   (*процесс*)
   IF "Technology".Regim = 11 THEN
       CASE "Technology".Regim_plan_stop_step OF
           0:  //плавный вывод ЗРГ на значение минимальной мощности ПИД регулятором
               IF "Sensors".ZRG_middle.Value THEN
                   "Control_ZRG".Mode := TRUE;
                   "Control_ZRG".Mode_from_PLC := TRUE;
                   IF "Control_ZRG".SP_PID > 10.0 THEN
                       "Control_ZRG".SP_PID := "Control_ZRG".SP_PID - 0.001;
                   END_IF;
               ELSE
                   //переход на следующий шаг
                   "Technology".Regim_plan_stop_step := 1;
               END_IF;

           1:  //Контроль достижения минимальной мощности
                   //снимаем защиту Понижение давления газа перед горелкой
                   "Alarms_and_warnings".Enable_Alarm_P_gas_before_burner_min := FALSE;
                   //снимаем защиту Повышение давления газа перед горелкой
                   "Alarms_and_warnings".Enable_Alarm_P_gas_before_burner_max := FALSE;
                   //отключаем ПИД регулирование ЗРГ
                   "Control_ZRG".Mode_from_PLC := FALSE;
                   "Control_ZRG".Manual_close_from_PLC := FALSE;
                   "Control_ZRG".Manual_open_from_PLC := FALSE;
                   //переход на следующий шаг
                   "Technology".Regim_plan_stop_step := 2;

           2:  //снимаем защиту Понижение давления сетевой воды за котлом
               "Alarms_and_warnings".Enable_Alarm_P_water_after_boiler_min := FALSE;
               //снимаем защиту Повышение давления сетевой воды за котлом
               "Alarms_and_warnings".Enable_Alarm_P_water_after_boiler_max := FALSE;
               //снимаем защиту Повышение температуры сетевой воды за котлом
               "Alarms_and_warnings".Enable_Alarm_T_water_after_boiler_max := FALSE;
               //снимаем защиту Понижение расхода сетевой воды через котел
               "Alarms_and_warnings".Enable_Alarm_Q_water_boiler_min := FALSE;

               //снимаем защиту Невоспламенение или погасание факела горелки котла
               "Alarms_and_warnings".Enable_Alarm_Not_flame_burner := FALSE;

               //перевод газовых исполнительных механизмов в исходное состояние
               "Control_PZK1".Mode := TRUE;    //закрываем ПЗК1
               "Control_PZK1".Avto_open := FALSE;
               "Control_PZK2".Mode := TRUE;    //закрываем ПЗК2
               "Control_PZK2".Avto_open := FALSE;
               "Control_KO".Mode := TRUE;  //закрываем КО
               "Control_KO".Avto_open := FALSE;
               "Control_KZ".Mode := TRUE;  //закрываем КЗ
               "Control_KZ".Avto_open := FALSE;
               "Control_KB".Mode := TRUE;  //открываем КБ
               "Control_KB".Avto_close := FALSE;
               "Control_IVN".Mode := TRUE; //отключаем ИВН
               "Control_IVN".Avto_on := FALSE;

               //перевод регуляторов разряжения и вентиляции на вентиляционные параметры
               IF "Sensors".DS_invertor_mode.Value THEN
                   "Control_DS".Mode := TRUE;
                   "Control_DS".Mode_from_PLC := TRUE;
                   "Control_DS".SP_PID := "RegMap".dP_furnace_ventilation;
               END_IF;
               IF "Sensors".DS_powergrid_mode.Value THEN
                   "Control_NAD".Mode := TRUE;
                   "Control_NAD".Mode_from_PLC := TRUE;
                   "Control_NAD".SP_PID := "RegMap".dP_furnace_ventilation;
               END_IF;
               IF "Sensors".DV_invertor_mode.Value THEN
                   "Control_DV".Mode := TRUE;
                   "Control_DV".Mode_from_PLC := TRUE;
                   "Control_DV".SP_PID := "RegMap".P_air_ventilation;
               END_IF;
               IF "Sensors".DV_powergrid_mode.Value THEN
                   "Control_NAV".Mode := TRUE;
                   "Control_NAV".Mode_from_PLC := TRUE;
                   "Control_NAV".SP_PID := "RegMap".P_air_ventilation;
               END_IF;

               //запускаем контрольный таймер
               "Timer".PLAN_STOP_temp_PT := T#60s;
               "Timer".PLAN_STOP_temp_IN := TRUE;
               //проверяем положение ИМ по газу
               IF NOT "Sensors".PZK1_open.Value AND
                   NOT "Sensors".PZK2_not_close.Value AND
                   NOT "Sensors".KO_open.Value AND
                   NOT "Sensors".KZ_open.Value AND
                   NOT "Sensors".KB_close.Value THEN
                   //переход далее
                   "Timer".PLAN_STOP_temp_IN := FALSE;
                   "Message".PLAN_STOP_not_initial_state_gas := FALSE;
                   "Technology".Regim_plan_stop_step := 3;
               END_IF;
               //если контрольное время вышло
               IF "Timer".PLAN_STOP_temp_Q THEN
                   "Message".PLAN_STOP_not_initial_state_gas := TRUE;
               END_IF;

           3:  //задержка 6 сек
               "Timer".PLAN_STOP_temp_PT := T#6s;
               "Timer".PLAN_STOP_temp_IN := TRUE;
               //переход далее
               IF "Timer".PLAN_STOP_temp_Q THEN
                   "Timer".PLAN_STOP_temp_IN := FALSE;
                   //переход на режим ПОСТОСТАНОВОЧНАЯ ОПРЕССОВКА
                   "Technology".Regim := 12;
               END_IF;
           ELSE
               "Technology".Regim_plan_stop_step := 0;
       END_CASE;
   ELSE
       //Сброс текущего шага
       "Technology".Regim_plan_stop_step := 0;
       //Сброс всех сообщений по данному режиму
       "Message".PLAN_STOP_not_initial_state_gas := FALSE;
       //сброс таймеров
       "Timer".PLAN_STOP_temp_IN := FALSE;
   END_IF;
END_FUNCTION

FUNCTION "Regim_STOP_PRESS" : Void   // FC22, SCL
{ S7_Optimized_Access := 'TRUE' }
VERSION : 0.1
BEGIN
   (*Режим ПОСТОСТАНОВОЧНАЯ ОПРЕССОВКА*)
   (*таймеры*)
   "Timer_STOP_PRESS_temp_DB".TON(IN := "Timer".STOP_PRESS_temp_IN,
                                  PT := "Timer".STOP_PRESS_temp_PT,
                                  Q => "Timer".STOP_PRESS_temp_Q);
   (*процесс*)
   IF "Technology".Regim = 12 THEN
       IF ("Sensors".DV_invertor_on.Value OR "Sensors".DV_powergrid_on.Value) AND
           ("Sensors".DS_invertor_on.Value OR "Sensors".DS_powergrid_on.Value) THEN
           CASE "Technology".Regim_stop_press_step OF
               0:  //анализ разрешения постостановочной опрессовки
                   IF "Technology".Stop_press_enable AND (NOT "Technology".Ventilation_conducted OR "Technology".transition_ignition) THEN
                       //переход на следующий шаг
                       "Technology".Regim_stop_press_step := 1;
                   ELSE
                       //переход на режим УКОРОЧЕННАЯ ВЕНТИЛЯЦИЯ
                       "Technology".Regim := 13;
                   END_IF;

               1:  //контроль положения исполнительных механизмов по газу
                   IF NOT "Sensors".PZK1_open.Value AND
                       NOT "Sensors".PZK2_not_close.Value AND
                       NOT "Sensors".KO_open.Value AND
                       NOT "Sensors".KZ_open.Value AND
                       NOT "Sensors".KB_close.Value THEN
                       //переход на следующий шаг
                       "Technology".Regim_stop_press_step := 2;
                   END_IF;

               2:  //контроль min P 
                   IF "Sensors".P_gas_before_PZK1_and_PZK2.Value < "Technology".SP_P_between_PZK_check_min THEN
                       //переход на следующий шаг
                       "Technology".Regim_stop_press_step := 3;
                   ELSE
                       "Message".STOP_PRESS_PZK1_or_KO_untight := TRUE;
                       "Technology".Regim_stop_press_step := 8;
                   END_IF;

               3:  //контроль max P
                   IF "Sensors".P_gas_before_PZK1_and_PZK2.Value < "Technology".SP_P_between_PZK_check_max THEN
                       //переход на следующий шаг
                       "Technology".Regim_stop_press_step := 4;
                   ELSE
                       "Message".STOP_PRESS_PZK1_or_KO_untight := TRUE;
                       "Technology".Regim_stop_press_step := 8;
                   END_IF;

               4:  //закрываем КБ
                   "Control_KB".Mode := TRUE;
                   "Control_KB".Avto_close := TRUE;
                   //контроль положения
                   IF "Sensors".KB_close.Value THEN
                       //переход на следующий шаг
                       "Timer".STOP_PRESS_temp_IN := FALSE;
                       "Technology".Regim_stop_press_step := 5;
                   END_IF;

               5:  //контроль отсутствия давления газа м/у ПЗК в течении заданного времени
                   "Timer".STOP_PRESS_temp_PT := T_CONV(INT_TO_DINT("Technology".SP_TIME_check_P_stop_press_min) * 1000);
                   "Timer".STOP_PRESS_temp_IN := TRUE;
                   IF "Timer".STOP_PRESS_temp_Q THEN
                       //переход на следующий шаг
                       "Timer".STOP_PRESS_temp_IN := FALSE;
                       "Technology".Regim_stop_press_step := 6;
                   ELSE
                       //если давление не в норме
                       IF ("Sensors".P_gas_before_PZK1_and_PZK2.Value > "Technology".SP_P_between_PZK_check_min) OR
                           ("Sensors".P_gas_before_PZK1_and_PZK2.Value > "Technology".SP_P_between_PZK_check_max) THEN
                           "Message".STOP_PRESS_PZK1_or_KO_untight := TRUE;
                           "Timer".STOP_PRESS_temp_IN := FALSE;
                           "Technology".Regim_stop_press_step := 8;
                       END_IF;
                   END_IF;

               6:  //открываем КО
                   "Control_KO".Mode := TRUE;
                   "Control_KO".Avto_open := TRUE;
                   IF "Sensors".KO_open.Value THEN
                       //переход на следующий шаг
                       "Timer".STOP_PRESS_temp_IN := FALSE;
                       "Technology".Regim_stop_press_step := 7;
                   END_IF;

               7:  //контроль достижения давления газа м/у ПЗК в течении заданного времени
                   "Timer".STOP_PRESS_temp_PT := T_CONV(INT_TO_DINT("Technology".SP_TIME_check_P_stop_press_max) * 1000);
                   "Timer".STOP_PRESS_temp_IN := TRUE;
                   IF "Timer".STOP_PRESS_temp_Q THEN
                       IF "Sensors".P_gas_before_BG_min.Value THEN
                           "Message".STOP_PRESS_P_before_BG_min := TRUE;
                       ELSE
                           "Message".STOP_PRESS_PZK2_or_KB_untight := TRUE;
                       END_IF;
                       "Timer".STOP_PRESS_temp_IN := FALSE;
                       "Technology".Regim_stop_press_step := 8;
                   ELSE
                       IF "Sensors".P_gas_before_PZK1_and_PZK2.Value > "Technology".SP_P_between_PZK_check_min THEN
                           //переход на следующий шаг
                           "Timer".STOP_PRESS_temp_IN := FALSE;
                           "Technology".Regim_stop_press_step := 8;
                       END_IF;
                   END_IF;

               8:  //закраваем КО
                   "Control_KO".Mode := TRUE;
                   "Control_KO".Avto_open := FALSE;
                   IF NOT "Sensors".KO_open.Value THEN
                       //переход на следующий шаг
                       "Technology".Regim_stop_press_step := 9;
                   END_IF;

               9:  //открываем КБ
                   "Control_KB".Mode := TRUE;
                   "Control_KB".Avto_close := FALSE;
                   IF NOT "Sensors".KB_close.Value THEN
                       //переход на следующий шаг
                       "Technology".Regim_stop_press_step := 10;
                   END_IF;

               10: //если опрессовка не прошла
                   IF "Message".STOP_PRESS_PZK1_or_KO_untight OR
                       "Message".STOP_PRESS_PZK2_or_KB_untight OR
                       "Message".STOP_PRESS_P_before_BG_min THEN
                       //переход на следующий шаг
                       "Timer".STOP_PRESS_temp_IN := FALSE;
                       "Technology".Regim_stop_press_step := 11;
                   ELSE
                       //если опрессовка успешно проведена
                       "Message".STOP_PRESS_success := TRUE;
                       //переход на следующий шаг
                       "Timer".STOP_PRESS_temp_IN := FALSE;
                       "Technology".Regim_stop_press_step := 11;
                   END_IF;

               11: //ожидание 5 сек
                   "Timer".STOP_PRESS_temp_PT := T#5s;
                   "Timer".STOP_PRESS_temp_IN := TRUE;
                   IF "Timer".STOP_PRESS_temp_Q THEN
                       "Timer".STOP_PRESS_temp_IN := FALSE;
                       "Message".STOP_PRESS_success := FALSE;
                       //переход на УКОРОЧЕННАЯ ВЕНТИЛЯЦИЯ
                       "Technology".Regim := 13;
                   END_IF;
               ELSE
                   "Technology".Regim_stop_press_step := 0;
           END_CASE;
       ELSE
           //перевод всех клапанов в исходное состояние
           "Control_PZK1".Mode := TRUE;        //закрываем ПЗК1
           "Control_PZK1".Avto_open := FALSE;
           "Control_PZK2".Mode := TRUE;        //закрываем ПЗК2
           "Control_PZK2".Avto_open := FALSE;
           "Control_KZ".Mode := TRUE;          //закрываем КЗ
           "Control_KZ".Avto_open := FALSE;
           "Control_KO".Mode := TRUE;          //закрываем КО
           "Control_KO".Avto_open := FALSE;
           "Control_KB".Mode := TRUE;          //открываем КБ
           "Control_KB".Avto_close := FALSE;
           "Control_IVN".Mode := TRUE;         //отключаем ИВН
           "Control_IVN".Avto_on := FALSE;
           //проверяем положение ИМ по газу
           IF NOT "Sensors".KB_close.Value AND //КБ открыт
               NOT "Sensors".KZ_open.Value AND //КЗ закрыт
               NOT "Sensors".KO_open.Value AND //КО закрыт
               NOT "Sensors".PZK1_open.Value AND   //ПЗК1 закрыт
               NOT "Sensors".PZK2_not_close.Value THEN  //ПЗК2 закрыт
               //переход далее
               //переход на УКОРОЧЕННАЯ ВЕНТИЛЯЦИЯ
               "Technology".Regim := 13;
           END_IF;
       END_IF;
   ELSE
       //сброс текущего шага
       "Technology".Regim_stop_press_step := 0;
       //сброс сообщений
       "Message".STOP_PRESS_PZK1_or_KO_untight := FALSE;
       "Message".STOP_PRESS_PZK2_or_KB_untight := FALSE;
       "Message".STOP_PRESS_P_before_BG_min := FALSE;
       "Message".STOP_PRESS_success := FALSE;
       //сброс таймеров
       "Timer".STOP_PRESS_temp_IN := FALSE;
   END_IF;
END_FUNCTION

FUNCTION "Regim_SHORT_VENTILATION" : Void   // FC23, SCL
{ S7_Optimized_Access := 'TRUE' }
VERSION : 0.1
BEGIN
   (*Режим УКОРОЧЕННАЯ ВЕНТИЛЯЦИЯ*)
   (*таймеры*)
   "Timer_SHORT_VENTILATION_temp_DB".TON(IN := "Timer".SHORT_VENTILATION_temp_IN,
                                         PT := "Timer".SHORT_VENTILATION_temp_PT,
                                         Q => "Timer".SHORT_VENTILATION_temp_Q);
   (*процесс*)
   IF "Technology".Regim = 13 THEN
       //снимаем защиту Повышение давления газа перед БГ
       "Alarms_and_warnings".Enable_Alarm_P_gas_before_BG_max := FALSE;
       //снимаем защиту Понижение давления газа перед БГ
       "Alarms_and_warnings".Enable_Alarm_P_gas_before_BG_min := FALSE;
       //закрываем ЗДГ
       "Control_ZDG".Mode := TRUE;
       "Control_ZDG".Avto_close := TRUE;
       "Control_ZDG".Avto_open := FALSE;
       "Control_ZDG".Avto_stop := FALSE;
       //разрешаем формирование предупреждения
       "Alarms_and_warnings".Enable_Warning_ZDG_not_close := TRUE;

       CASE "Technology".Regim_short_ventilation_step OF
           0:  //снимаем защиту Понижение давления воздуха перед горелкой
               "Alarms_and_warnings".Enable_Alarm_P_air_before_burner_min := FALSE;
               //снимаем защиту Понижение разряжения в топке
               "Alarms_and_warnings".Enable_Alarm_dP_furnace_boiler_min := FALSE;
               "Technology".Regim_short_ventilation_step := 1;
           1:
               IF (("Sensors".DS_invertor_mode.Value AND "Sensors".DS_invertor_on.Value) AND
                   "Control_DS".Mode = TRUE AND
                   "Control_DS".Mode_from_PLC = TRUE AND
                   "Control_DS".SP_PID = "RegMap".dP_furnace_ventilation) OR
                   (("Sensors".DS_powergrid_mode.Value AND "Sensors".DS_powergrid_on.Value) AND
                   "Control_NAD".Mode = TRUE AND
                   "Control_NAD".Mode_from_PLC = TRUE AND
                   "Control_NAD".SP_PID = "RegMap".dP_furnace_ventilation) THEN
                   //переход через шаг
                   "Timer".SHORT_VENTILATION_temp_IN := FALSE;
                   "Technology".Regim_short_ventilation_step := 3;
               ELSE
                   //переход на поддержание вентиляционного значения разряжения    
                   //если работаем от ПЧ
                   IF ("Sensors".DS_invertor_mode.Value AND "Sensors".DS_invertor_on.Value) THEN
                       "Control_DS".Mode := TRUE;
                       "Control_DS".Mode_from_PLC := TRUE;
                       "Control_DS".SP_PID := "RegMap".dP_furnace_ventilation;
                   END_IF;
                   //если работаем от сети
                   IF ("Sensors".DS_powergrid_mode.Value AND "Sensors".DS_powergrid_on.Value) THEN
                       "Control_NAD".Mode := TRUE;
                       "Control_NAD".Mode_from_PLC := TRUE;
                       "Control_NAD".SP_PID := "RegMap".dP_furnace_ventilation;
                   END_IF;
                   //переход на следующий шаг
                   "Timer".SHORT_VENTILATION_temp_IN := FALSE;
                   "Technology".Regim_short_ventilation_step := 2;
               END_IF;

           2:  //ожидание 6 сек
                   "Timer".SHORT_VENTILATION_temp_PT := T#6s;
                   "Timer".SHORT_VENTILATION_temp_IN := TRUE;
                   IF "Timer".SHORT_VENTILATION_temp_Q THEN
                       "Timer".SHORT_VENTILATION_temp_IN := FALSE;
                       //переход на следующий шаг
                       "Technology".Regim_short_ventilation_step := 3;
                   END_IF;

           3:  //переход на поддержание вентиляционного значения давления воздуха
               //если работаем от ПЧ
               IF ("Sensors".DV_invertor_mode.Value AND "Sensors".DV_invertor_on.Value) THEN
                   "Control_DV".Mode := TRUE;
                   "Control_DV".Mode_from_PLC := TRUE;
                   "Control_DV".SP_PID := "RegMap".P_air_ventilation;
                   //переход на следующий шаг 
                   "Timer".SHORT_VENTILATION_temp_IN := FALSE;
                   "Technology".Regim_short_ventilation_step := 4;
               END_IF;
               //если ДВ работает от сети, то НАВ открываем до среднего положения
               IF ("Sensors".DV_powergrid_mode.Value AND "Sensors".DV_powergrid_on.Value) THEN
                   "Control_NAV".Mode := TRUE;
                   "Control_NAV".Mode_from_PLC := FALSE;
                   IF NOT "Sensors".NAV_middle.Value THEN
                       "Control_NAV".Manual_open_from_PLC := TRUE;
                   ELSE
                       "Control_NAV".Manual_open_from_PLC := FALSE;
                       //переход на следующий шаг 
                       "Timer".SHORT_VENTILATION_temp_IN := FALSE;
                       "Technology".Regim_short_ventilation_step := 4;
                   END_IF;
               END_IF;

           4:  //анализ разрешения проведения укороченной вентиляции
               IF "Technology".Short_ventilation_enable AND NOT "Technology".Ventilation_conducted THEN
                   //запускаем таймер укороченной вентиляции
                   "Timer".SHORT_VENTILATION_temp_PT := T_CONV(INT_TO_DINT("Technology".SP_TIME_Short_ventilation) * 1000);
                   "Timer".SHORT_VENTILATION_temp_IN := TRUE;
                   IF "Timer".SHORT_VENTILATION_temp_Q THEN
                       "Timer".SHORT_VENTILATION_temp_IN := FALSE;
                       //переход на следующий шаг
                       "Message".SHORT_VENTILATION_ok := TRUE;
                       //переход в режим ОЖИДАНИЕ 
                       "Technology".Regim := 1;
                       "Technology".Regim_off_step := 1;
                       //"Technology".Regim_short_ventilation_step := 5;
                   END_IF;
               ELSE
                   "Timer".SHORT_VENTILATION_temp_IN := FALSE;
                   //переход в режим ОЖИДАНИЕ 
                   "Technology".Regim := 1;
                   "Technology".Regim_off_step := 1;
               END_IF;

   (*        5:  //переход на поддержание розжигового значения разряжения
               //если работаем от ПЧ
               IF ("Sensors".DS_invertor_mode.Value AND "Sensors".DS_invertor_on.Value) THEN
                   "Control_DS".Mode := TRUE;
                   "Control_DS".Mode_from_PLC := TRUE;
                   "Control_DS".SP_PID := "RegMap".dP_furnace_ignition;
               END_IF;
               //если работаем от сети
               IF ("Sensors".DS_powergrid_mode.Value AND "Sensors".DS_powergrid_on.Value) THEN
                   "Control_NAD".Mode := TRUE;
                   "Control_NAD".Mode_from_PLC := TRUE;
                   "Control_NAD".SP_PID := "RegMap".dP_furnace_ignition;
               END_IF;
               //переход на следующий шаг
               "Timer".SHORT_VENTILATION_temp_IN := FALSE;
               "Technology".Regim_short_ventilation_step := 6;

           6:  //ожидание 6 сек
               "Timer".SHORT_VENTILATION_temp_PT := T#6s;
               "Timer".SHORT_VENTILATION_temp_IN := TRUE;
               IF "Timer".SHORT_VENTILATION_temp_Q THEN
                   "Timer".SHORT_VENTILATION_temp_IN := FALSE;
                   //переход на следующий шаг
                   "Technology".Regim_short_ventilation_step := 7;
               END_IF;

           7:  //переход на поддержание розжигового значения давления воздуха
               //если работаем от ПЧ
               IF ("Sensors".DV_invertor_mode.Value AND "Sensors".DV_invertor_on.Value) THEN
                   "Control_DV".Mode := TRUE;
                   "Control_DV".Mode_from_PLC := TRUE;
                   "Control_DV".SP_PID := "RegMap".P_air_ignition;
               END_IF;
               //если работает от сети
               IF ("Sensors".DV_powergrid_mode.Value AND "Sensors".DV_powergrid_on.Value) THEN
                   "Control_NAV".Mode := TRUE;
                   "Control_NAV".Mode_from_PLC := TRUE;
                   "Control_NAV".SP_PID := "RegMap".P_air_ignition;
               END_IF;
               //переход в режим ОЖИДАНИЕ 
               "Technology".Regim := 1;
               "Technology".Regim_off_step := 1;*)
           ELSE
               "Technology".Regim_short_ventilation_step := 0;
       END_CASE;

       IF NOT "Sensors".DV_invertor_on.Value AND NOT "Sensors".DV_powergrid_on.Value AND NOT "Sensors".DS_invertor_on.Value AND NOT "Sensors".DS_powergrid_on.Value AND
           (NOT "Sensors".ZDG_no_close.Value OR "Alarms_and_warnings".Enable_Warning_ZDG_not_close) THEN
           //переход на режим ОТКЛ
           "Technology".Regim := 1;
           "Technology".Regim_off_step := 2;
       END_IF;
   ELSE
       //сброс текущего шага
       "Technology".Regim_short_ventilation_step := 0;
       //сброс сообщений
       "Message".SHORT_VENTILATION_ok := FALSE;
       //сброс таймеров
       "Timer".SHORT_VENTILATION_temp_IN := FALSE;
       //снимаем предупреждение
       "Alarms_and_warnings".Enable_Warning_ZDG_not_close := FALSE;
   END_IF;
END_FUNCTION

FUNCTION "Regim_TEST_PRESS" : Void   // FC27, SCL
{ S7_Optimized_Access := 'TRUE' }
VERSION : 0.1
BEGIN
   (*Режим ТЕСТОВАЯ ОПРЕССОВКА*)
   (*таймеры*)
   (*процесс*)
   IF "Technology".Regim = 14 THEN
       CASE "Technology".Regim_test_press_step OF
           0:
               ;
           ELSE
               "Technology".Regim_test_press_step := 0;
       END_CASE;
   ELSE
       //Сброс текущего шага
       "Technology".Regim_test_press_step := 0;
       //Сброс всех сообщений по данному режиму
       //сброс таймеров
   END_IF;
END_FUNCTION

FUNCTION "Regim_TEST_IGNITION" : Void   // FC28, SCL
{ S7_Optimized_Access := 'TRUE' }
VERSION : 0.1
BEGIN
   (*Режим РОЗЖИГ*)
   (*таймеры*)
   (*процесс*)
   IF "Technology".Regim = 15 THEN
       CASE "Technology".Regim_test_ignition_step OF
           0:
               ;
           ELSE
               "Technology".Regim_test_ignition_step := 0;
       END_CASE;
   ELSE
       //сброс текущего шага
       "Technology".Regim_test_ignition_step := 0;
       //сброс сообщений
       //сброс таймеров
   END_IF;
END_FUNCTION